(* CoDeSys 2.3.9.35 project: Сушка v1.1.pro *)
(* Libraries: IECSFC.LIB 13.4.06 15:51:28, ANALYZATION.LIB 5.10.99 09:05:06, Util.lib 18.5.10 15:14:28, STANDARD.LIB 4.10.05 11:14:46, SYSLIBTIME.LIB 20.2.06 13:31:16 *)

(* PLC configuration (modules and I/O channels)
Fast discrete inputs [I_SIMPLE_INPUT] node 0, in %IB0 out %QB0 {Filtrationtime = 10; Visibility = No}
  AT %IX0.0 [BitInput] Discrete input 1
  AT %IX0.1 [BitInput] Discrete input 2
Discrete inputs - 16 [ID130] node 1, in %IB1 out %QB1 {Filtrationtime_GeneralINP = 1; Visibility = No; PinCount = 16}
  AT %IB1.0 [ByteInput] 8 discrete inputs
  AT %IB1.1 [ByteInput] 8 discrete inputs
Fast discrete outputs [OWEN_ID570] node 2, in %IB2 out %QB2 {SafeValueBool = FALSE; SafeValueBool = FALSE; SafeValueBool = FALSE; SafeValueBool = FALSE; Visibility = No}
  AT %QX2.0 [BitOutput] Fast discrete output 1
  AT %QX2.1 [BitOutput] Fast discrete output 2
  AT %QX2.2 [BitOutput] Fast discrete output 3
  AT %QX2.3 [BitOutput] Fast discrete output 4
Discrete outputs - 8 [ID131] node 3, in %IB3 out %QB3 {SafeValueByte = 0; Visibility = No; PinCount = 10}
  AT %QB3.0 [ByteOutput] 8 discrete outputs
Special input [ID103] node 4, in %IB4 out %QB4 {Filtrationtime = 1000; PinCount = 1; WatchDogPeriod = 400; PollPeriod = 3000; Visibility = No}
  AT %IX4.0 [BitInput] Special input
Special output [ID104] node 5, in %IB5 out %QB5 {Visibility = No; PinCount = 1}
  AT %QX5.0 [BitOutput] Special output
AT %QD6.0 [DWordOutput] Last address
AT %QW6.1 [WordOutput] Last error
RS-485-1 [COM1_USART] node 0, in %IB6.0 out %QB6.0 {CommunicationSpeed = 9600; Parity = NO PARITY CHECK; BitLength = 8 bits; StopLength = One stop bit; InterfaceType = RS485; FrameOriented = RTU; Timeout = 0; Visibility = No}
AT %QB6.1.0 [ComChannel] Command (0xff - Start)
AT %IW6.1.0.0 [WordInput]
AT %IW6.1.1.0 [WordInput]
AT %IW6.1.2.0 [WordInput]
Button [ID003] node 7, in %IB7 out %QB7
  AT %IX7.0 [BitInput] Button Start/Stop
RS-485-2 [COM3_USART] node 0, in %IB8.0.0 out %QB8.0.0 {CommunicationSpeed = 11520; Parity = NO PARITY CHECK; BitLength = 8 bits; StopLength = One stop bit; InterfaceType = RS232; FrameOriented = RTU; Timeout = 0; Visibility = No}
TCP [TCP_ID221] node 1, in %IB8.0.1 out %QB8.0.1 {RemotePort = 502; Visibility = No}
2 byte [Register] node 1, in %IB8.1 out %QB8.1
  AT %QW8.1.0 [WordOutput]
2 byte [Register] node 2, in %IB8.2 out %QB8.2
  AT %QW8.2.0 [WordOutput]
2 byte [Register] node 3, in %IB8.3 out %QB8.3
  AT %QW8.3.0 [WordOutput]
2 byte [Register] node 4, in %IB8.4 out %QB8.4
  AT %QW8.4.0 [WordOutput]
2 byte [Register] node 5, in %IB8.5 out %QB8.5
  AT %QW8.5.0 [WordOutput]
2 byte [Register] node 6, in %IB8.6 out %QB8.6
  AT %QW8.6.0 [WordOutput]
2 byte [Register] node 7, in %IB8.7 out %QB8.7
  AT %QW8.7.0 [WordOutput]
2 byte [Register] node 8, in %IB8.8 out %QB8.8
  AT %QW8.8.0 [WordOutput]
2 byte [Register] node 9, in %IB8.9 out %QB8.9
  AT %QW8.9.0 [WordOutput]
2 byte [Register] node 10, in %IB8.10 out %QB8.10
  AT %QW8.10.0 [WordOutput]
2 byte [Register] node 11, in %IB8.11 out %QB8.11
  AT %QW8.11.0 [WordOutput]
2 byte [Register] node 12, in %IB8.12 out %QB8.12
  AT %QW8.12.0 [WordOutput]
2 byte [Register] node 13, in %IB8.13 out %QB8.13
  AT %QW8.13.0 [WordOutput]
2 byte [Register] node 14, in %IB8.14 out %QB8.14
  AT %QW8.14.0 [WordOutput]
2 byte [Register] node 15, in %IB8.15 out %QB8.15
  AT %QW8.15.0 [WordOutput]
2 byte [Register] node 16, in %IB8.16 out %QB8.16
  AT %QW8.16.0 [WordOutput]
2 byte [Register] node 17, in %IB8.17 out %QB8.17
  AT %QW8.17.0 [WordOutput]
2 byte [Register] node 18, in %IB8.18 out %QB8.18
  AT %QW8.18.0 [WordOutput]
2 byte [Register] node 19, in %IB8.19 out %QB8.19
  AT %QW8.19.0 [WordOutput]
2 byte [Register] node 20, in %IB8.20 out %QB8.20
  AT %QW8.20.0 [WordOutput]
  AT %QW8.21.0 [WordOutput]
  AT %QW8.22.0 [WordOutput]
  AT %QW8.23.0 [WordOutput]
  AT %QW8.24.0 [WordOutput]
  AT %QW8.25.0 [WordOutput]
  AT %QW8.26.0 [WordOutput]
AT %QB8.27.0 [ByteOutput]
AT %QW8.28.0 [WordOutput]
AT %QW8.29.0 [WordOutput]
AT %QW8.30.0 [WordOutput]
AT %QW8.31.0 [WordOutput]
*)

(* POU PLC_PRG, LD *)
PROGRAM PLC_PRG
VAR
(* Блок часов реального времени*)
	get_time: t_n_d;
	outSecond: WORD;
	outMinute AT %QW8.26.0: WORD;
	outHour AT %QW8.25.0: WORD;
	outDay AT %QW8.24.0: WORD;
	outMonth AT %QW8.13.0: WORD;
	outYear AT %QW8.14.0: WORD;
	outDayOfWeek: WORD;
(*Насторойка часов реального времени*)
	inMin AT %QW8.10.0:WORD;
	inHour AT %QW8.11.0:WORD;
	inday AT %QW8.12.0:WORD;
(*Команда на старт определенной печи по заданному времени*)
	Start1: BOOL;
	Start2: BOOL;
	Start3: BOOL;
(*Команда на остановку определенной печи через промежуток времени, заданный оператором*)
	stop1: BOOL;
	stop2: BOOL;
	stop3: BOOL;
(*Блоки-регуляторы включения\отключения вентиляторов и тенов, в зависимости от темпреатуры*)
	HYST1: HYSTERESIS;
	min_temp1: WORD;
	max_temp1: WORD;
	out1: BOOL;
	HYST2: HYSTERESIS;
	max_temp2: WORD;
	min_temp2: WORD;
	out2: BOOL;
	HYST3: HYSTERESIS;
	max_temp3: WORD;
	min_temp3: WORD;
	out3: BOOL;
(*Блоки задания на влючение, в зависимости от реального времени*)
	set_time_start1: s_t_s;
	set_time_start2: s_t_s;
	set_time_start3: s_t_s;
(*Продолжительность сушки после достижения номинальной температуры*)
	time_stop1: t_stop;
	time_stop2: t_stop;
	time_stop3: t_stop;
(*Входящая температура*)
	in_temp1 AT %IW6.1.0.0: WORD;
	in_temp2 AT %IW6.1.1.0: WORD;
	in_temp3 AT %IW6.1.2.0: WORD;
(*Блок для упрощения схемы*)
	min_max: min_max;
(*Выходные сигналы для управления вентиляторами и тенами*)
	vent1 AT %QX2.3: BOOL;
	vent2 AT %QX3.0.1: BOOL;
	vent3 AT %QX3.0.3: BOOL;

	ten1 AT %QX2.2: BOOL;
	ten2 AT %QX3.0.0: BOOL;
	ten3 AT %QX3.0.2: BOOL;

	ton1: TON;
	ton2: TON;
	ton3: TON;

(*Входной переключатель автомат/ручное*)
	in_switch1 AT %IX0.0:BOOL;
(*Выходное отображение автомат/ручное*)
	in_sw1 AT %QX8.27.0.0:BOOL;
(*Выходящая температура для отображения*)
	out_temp1 AT %QW8.21.0: WORD;
	out_temp2 AT %QW8.22.0: WORD;
	out_temp3 AT %QW8.23.0: WORD;
(*Параметры вносимые оператором для блока задания на влючение печи сушки №1*)
	Hour_IP1 AT %QW8.1.0: WORD;
	Minute_IP1 AT %QW8.2.0: WORD;
	Day_IP1 AT %QW8.3.0: WORD;
(*Параметры вносимые оператором для блока задания на влючение печи сушки №2*)
	Hour_IP2 AT %QW8.4.0: WORD;
	Minute_IP2 AT %QW8.5.0: WORD;
	Day_IP2 AT %QW8.6.0: WORD;
(*Параметры вносимые оператором для блока задания на влючение печи сушки №3*)
	Hour_IP3 AT %QW8.7.0: WORD;
	Minute_IP3 AT %QW8.8.0: WORD;
	Day_IP3 AT %QW8.9.0: WORD;
(*Время работы, вносимые оператором для печей сушек №1,2,3*)
	work_time1 AT %QW8.15.0: WORD;
	work_time2 AT %QW8.16.0: WORD;
	work_time3 AT %QW8.17.0: WORD;
(*Уставки температуры, вносимые оператором для печей сушек №1,2,3*)
	set_temp1 AT %QW8.18.0: WORD;
	set_temp2 AT %QW8.19.0: WORD;
	set_temp3 AT %QW8.20.0: WORD;
(*Выходное отображение старта системы*)
	Start11 AT %QX8.27.0.1: BOOL;
	Start22 AT %QX8.27.0.2: BOOL;
	Start33 AT %QX8.27.0.3: BOOL;
(*Кнопка подтверддения пуска*)
	but_in1 AT %QW8.28.0:WORD;
	but1: BOOL;
	but_in2 AT %QW8.29.0:WORD;
	but2: BOOL;
	but_in3 AT %QW8.30.0:WORD;
	but3: BOOL;
(*Кнопка "Грибок"*)
	stop_grib AT %IX0.1: BOOL;
(*Контроль аварийного привышения температуры в камерах сушил №1,2,3*)
	av_1 AT %IX1.0.0: BOOL;
	av_2 AT %IX1.0.1: BOOL;
	av_3 AT %IX1.0.2: BOOL;
(*Коменда установки значений RTC*)
	set_t:BOOL;
(*Выходное реле выбора режима работы*)
	avto_ruch AT %QX2.1: BOOL;
(*Блок остановки программы по приходу нуля из Scada&*)
	stop_if: stop_if;
	st_if1: BOOL;
	st_if2: BOOL;
	st_if3: BOOL;

	set_time AT %QW8.31.0: WORD;
END_VAR
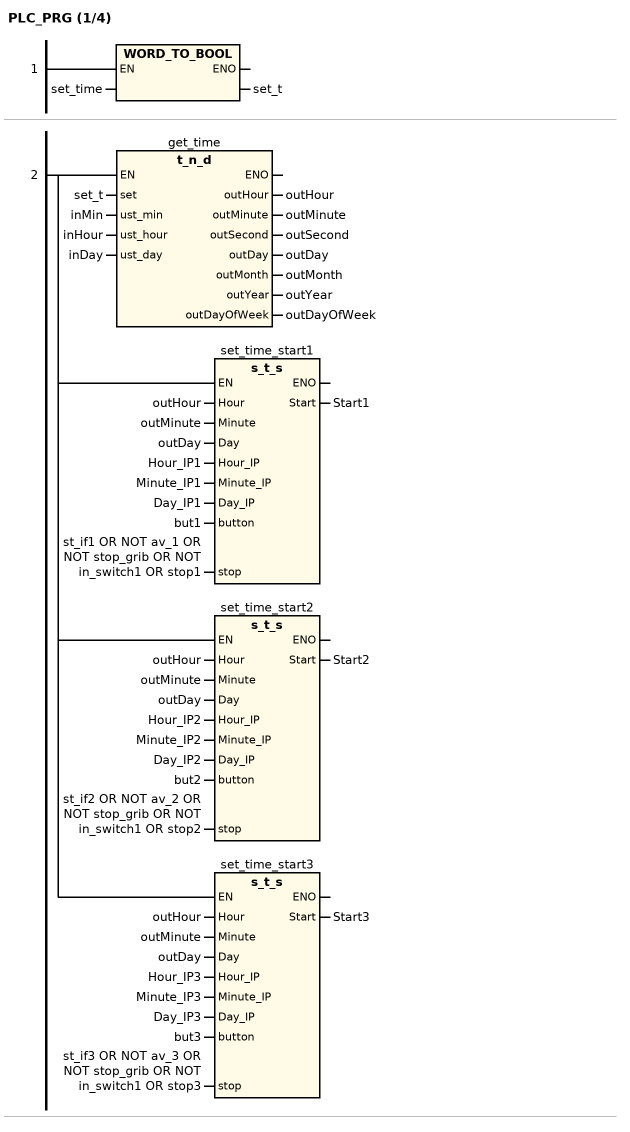
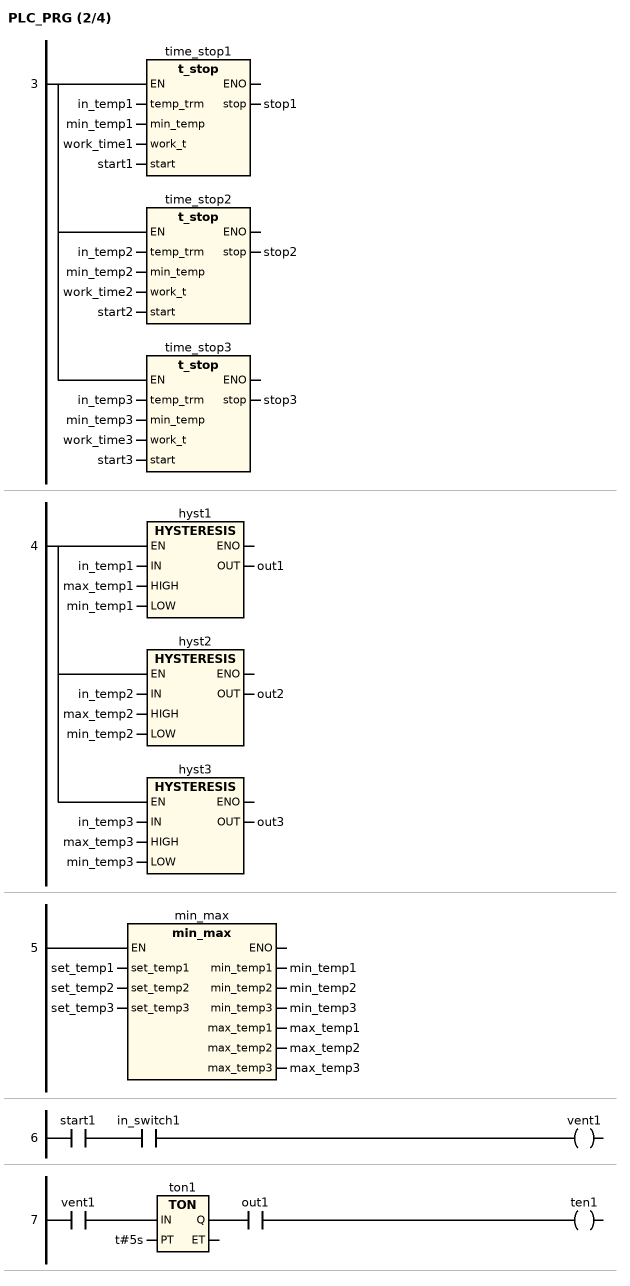
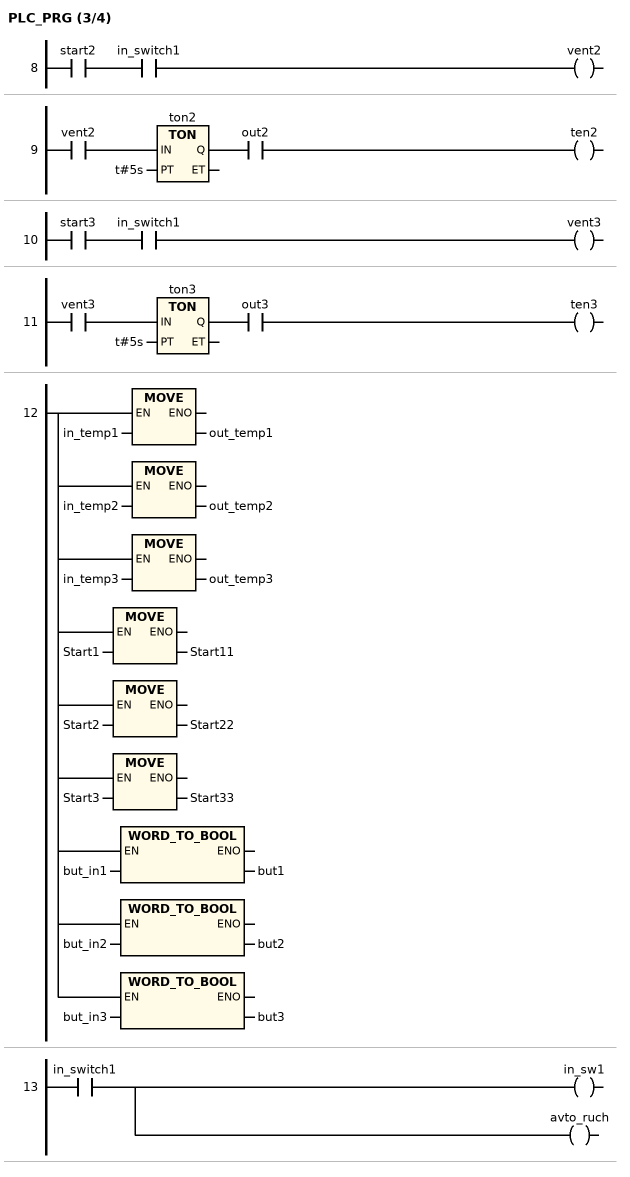
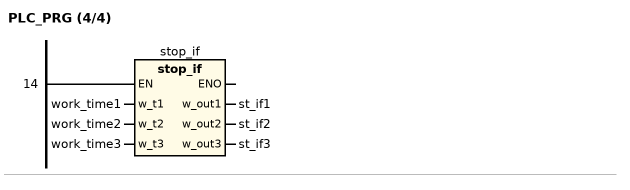
_LD_ (* Ladder Diagram *)
NETWORK 1
	*
		EN --- WORD_TO_BOOL(set_time) => set_t
NETWORK 2
	*
		EN --- get_time:t_n_d(set: set_t, ust_min: inMin, ust_hour: inHour, ust_day: inDay, outMinute => outMinute, outSecond => outSecond, outDay => outDay, outMonth => outMonth, outYear => outYear, outDayOfWeek => outDayOfWeek) => outHour
		EN --- set_time_start1:s_t_s(Hour: outHour, Minute: outMinute, Day: outDay, Hour_IP: Hour_IP1, Minute_IP: Minute_IP1, Day_IP: Day_IP1, button: but1, stop: st_if1 OR NOT av_1 OR NOT stop_grib OR NOT in_switch1 OR stop1) => Start1
		EN --- set_time_start2:s_t_s(Hour: outHour, Minute: outMinute, Day: outDay, Hour_IP: Hour_IP2, Minute_IP: Minute_IP2, Day_IP: Day_IP2, button: but2, stop: st_if2 OR NOT av_2 OR NOT stop_grib OR NOT in_switch1 OR stop2) => Start2
		EN --- set_time_start3:s_t_s(Hour: outHour, Minute: outMinute, Day: outDay, Hour_IP: Hour_IP3, Minute_IP: Minute_IP3, Day_IP: Day_IP3, button: but3, stop: st_if3 OR NOT av_3 OR NOT stop_grib OR NOT in_switch1 OR stop3) => Start3
NETWORK 3
	*
		EN --- time_stop1:t_stop(temp_trm: in_temp1, min_temp: min_temp1, work_t: work_time1, start: start1) => stop1
		EN --- time_stop2:t_stop(temp_trm: in_temp2, min_temp: min_temp2, work_t: work_time2, start: start2) => stop2
		EN --- time_stop3:t_stop(temp_trm: in_temp3, min_temp: min_temp3, work_t: work_time3, start: start3) => stop3
NETWORK 4
	*
		EN --- hyst1:HYSTERESIS(IN: in_temp1, HIGH: max_temp1, LOW: min_temp1) => out1
		EN --- hyst2:HYSTERESIS(IN: in_temp2, HIGH: max_temp2, LOW: min_temp2) => out2
		EN --- hyst3:HYSTERESIS(IN: in_temp3, HIGH: max_temp3, LOW: min_temp3) => out3
NETWORK 5
	*
		EN --- min_max:min_max(set_temp1: set_temp1, set_temp2: set_temp2, set_temp3: set_temp3, min_temp2 => min_temp2, min_temp3 => min_temp3, max_temp1 => max_temp1, max_temp2 => max_temp2, max_temp3 => max_temp3) => min_temp1
NETWORK 6
	[start1] - [in_switch1] --- (vent1)
NETWORK 7
	[vent1] - ton1:TON(IN: *, PT: t#5s) - [out1] --- (ten1)
NETWORK 8
	[start2] - [in_switch1] --- (vent2)
NETWORK 9
	[vent2] - ton2:TON(IN: *, PT: t#5s) - [out2] --- (ten2)
NETWORK 10
	[start3] - [in_switch1] --- (vent3)
NETWORK 11
	[vent3] - ton3:TON(IN: *, PT: t#5s) - [out3] --- (ten3)
NETWORK 12
	*
		EN --- MOVE(in_temp1) => out_temp1
		EN --- MOVE(in_temp2) => out_temp2
		EN --- MOVE(in_temp3) => out_temp3
		EN --- MOVE(Start1) => Start11
		EN --- MOVE(Start2) => Start22
		EN --- MOVE(Start3) => Start33
		EN --- WORD_TO_BOOL(but_in1) => but1
		EN --- WORD_TO_BOOL(but_in2) => but2
		EN --- WORD_TO_BOOL(but_in3) => but3
NETWORK 13
	[in_switch1] --- (in_sw1) (avto_ruch)
NETWORK 14
	*
		EN --- stop_if:stop_if(w_t1: work_time1, w_t2: work_time2, w_t3: work_time3, w_out2 => st_if2, w_out3 => st_if3) => st_if1
_END_LD_
(* the same logic as Structured Text *)
(* Network 1 *)
set_t := WORD_TO_BOOL(set_time);
(* Network 2 *)
get_time(set := set_t, ust_min := inMin, ust_hour := inHour, ust_day := inDay);
outMinute := get_time.outMinute;
outSecond := get_time.outSecond;
outDay := get_time.outDay;
outMonth := get_time.outMonth;
outYear := get_time.outYear;
outDayOfWeek := get_time.outDayOfWeek;
outHour := get_time.outHour;
set_time_start1(Hour := outHour, Minute := outMinute, Day := outDay, Hour_IP := Hour_IP1, Minute_IP := Minute_IP1, Day_IP := Day_IP1, button := but1, stop := st_if1 OR NOT av_1 OR NOT stop_grib OR NOT in_switch1 OR stop1);
Start1 := set_time_start1.Start;
set_time_start2(Hour := outHour, Minute := outMinute, Day := outDay, Hour_IP := Hour_IP2, Minute_IP := Minute_IP2, Day_IP := Day_IP2, button := but2, stop := st_if2 OR NOT av_2 OR NOT stop_grib OR NOT in_switch1 OR stop2);
Start2 := set_time_start2.Start;
set_time_start3(Hour := outHour, Minute := outMinute, Day := outDay, Hour_IP := Hour_IP3, Minute_IP := Minute_IP3, Day_IP := Day_IP3, button := but3, stop := st_if3 OR NOT av_3 OR NOT stop_grib OR NOT in_switch1 OR stop3);
Start3 := set_time_start3.Start;
(* Network 3 *)
time_stop1(temp_trm := in_temp1, min_temp := min_temp1, work_t := work_time1, start := start1);
stop1 := time_stop1.stop;
time_stop2(temp_trm := in_temp2, min_temp := min_temp2, work_t := work_time2, start := start2);
stop2 := time_stop2.stop;
time_stop3(temp_trm := in_temp3, min_temp := min_temp3, work_t := work_time3, start := start3);
stop3 := time_stop3.stop;
(* Network 4 *)
hyst1(IN := in_temp1, HIGH := max_temp1, LOW := min_temp1);
out1 := hyst1.OUT;
hyst2(IN := in_temp2, HIGH := max_temp2, LOW := min_temp2);
out2 := hyst2.OUT;
hyst3(IN := in_temp3, HIGH := max_temp3, LOW := min_temp3);
out3 := hyst3.OUT;
(* Network 5 *)
min_max(set_temp1 := set_temp1, set_temp2 := set_temp2, set_temp3 := set_temp3);
min_temp2 := min_max.min_temp2;
min_temp3 := min_max.min_temp3;
max_temp1 := min_max.max_temp1;
max_temp2 := min_max.max_temp2;
max_temp3 := min_max.max_temp3;
min_temp1 := min_max.min_temp1;
(* Network 6 *)
vent1 := start1 AND in_switch1;
(* Network 7 *)
ton1(IN := vent1, PT := t#5s);
ten1 := ton1.Q AND out1;
(* Network 8 *)
vent2 := start2 AND in_switch1;
(* Network 9 *)
ton2(IN := vent2, PT := t#5s);
ten2 := ton2.Q AND out2;
(* Network 10 *)
vent3 := start3 AND in_switch1;
(* Network 11 *)
ton3(IN := vent3, PT := t#5s);
ten3 := ton3.Q AND out3;
(* Network 12 *)
out_temp1 := in_temp1;
out_temp2 := in_temp2;
out_temp3 := in_temp3;
Start11 := Start1;
Start22 := Start2;
Start33 := Start3;
but1 := WORD_TO_BOOL(but_in1);
but2 := WORD_TO_BOOL(but_in2);
but3 := WORD_TO_BOOL(but_in3);
(* Network 13 *)
in_sw1 := in_switch1;
avto_ruch := in_switch1;
(* Network 14 *)
stop_if(w_t1 := work_time1, w_t2 := work_time2, w_t3 := work_time3);
st_if2 := stop_if.w_out2;
st_if3 := stop_if.w_out3;
st_if1 := stop_if.w_out1;
END_PROGRAM

(* POU t_n_d, ST *)
FUNCTION_BLOCK t_n_d
VAR
	GetTime: CurTimeEx;
	TimeAndDate: SystemTimeDate;
	Sys_Time: SysTime64;
END_VAR

VAR_INPUT
	set: BOOL;
	ust_min:WORD;
	ust_hour:WORD;
	ust_day:WORD;
END_VAR

VAR_OUTPUT
	outHour: WORD;
	outMinute: WORD;
	outSecond: WORD;
	outDay: WORD;
	outMonth: WORD;
	outYear: WORD;
	outDayOfWeek: WORD;
END_VAR
(*Текущее время*)
	TimeAndDate.Day :=0;
	TimeAndDate.DayOfWeek :=0;
	TimeAndDate.dwHighMsec :=0;
	TimeAndDate.dwLowMSecs :=0;
	TimeAndDate.Milliseconds :=0;
	TimeAndDate.Minute :=0;
	TimeAndDate.Second :=0;
	TimeAndDate.Hour :=0;
	TimeAndDate.Year :=0;
	TimeAndDate.Month :=0;
	Sys_time.ulHigh :=0;
	Sys_time.ulLow :=0;
	GetTime (SystemTime:=Sys_Time , TimeDate:= TimeAndDate);

IF set THEN
	TimeAndDate.Day :=ust_day;
	TimeAndDate.Minute :=ust_min;
	TimeAndDate.Hour :=ust_hour;
	GetTime (SystemTime:=Sys_Time , TimeDate:= TimeAndDate);
END_IF

	outSecond:=TimeAndDate.Second;
	outMinute:=TimeAndDate.Minute;
	outHour:=TimeAndDate.Hour;
	outDay:=TimeAndDate.Day;
	outMonth:=TimeAndDate.Month;
	outYear:=TimeAndDate.Year;
	outDayOfWeek:=TimeAndDate.DayOfWeek;

(*	outdwHighMsec:=TimeAndDate.dwHighMsec;
	outdwLowMSecs:=TimeAndDate.dwLowMSecs;*)

(*	outulHigh:=Sys_time.ulHigh;
	outulLow:=Sys_time.ulLow;*)
END_FUNCTION_BLOCK

(* POU s_t_s, LD *)
FUNCTION_BLOCK s_t_s

VAR_INPUT
	Hour: WORD;
	Minute: WORD;
	Day: WORD;
	Hour_IP: WORD;
	Minute_IP: WORD;
	Day_IP: WORD;
	button: BOOL;
	stop: BOOL;
END_VAR
VAR
	set_hour: BOOL;
	set_min: BOOL;
	set_day: BOOL;
	r_t: R_TRIG;
	pr1: BOOL;
	pr2: BOOL;
END_VAR
VAR_OUTPUT
	Start: BOOL;
END_VAR
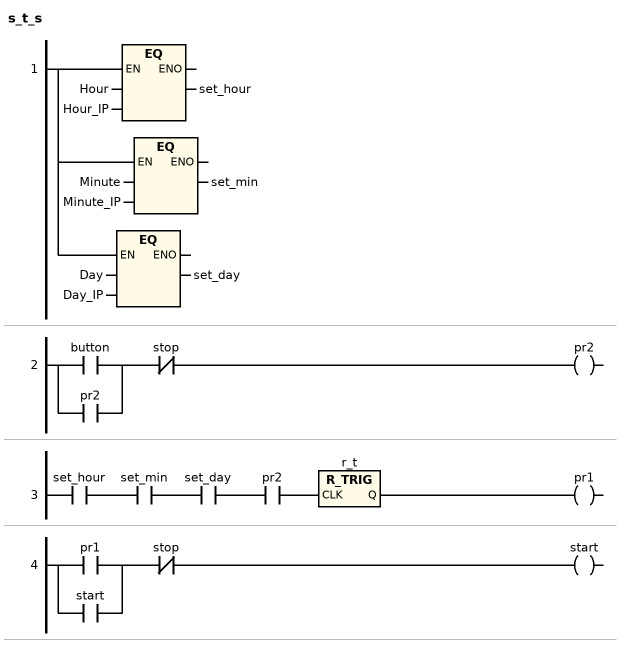
_LD_ (* Ladder Diagram *)
NETWORK 1
	*
		EN --- EQ(Hour, Hour_IP) => set_hour
		EN --- EQ(Minute, Minute_IP) => set_min
		EN --- EQ(Day, Day_IP) => set_day
NETWORK 2
	{ [button] | [pr2] } - [/stop] --- (pr2)
NETWORK 3
	[set_hour] - [set_min] - [set_day] - [pr2] - r_t:R_TRIG(CLK: *) --- (pr1)
NETWORK 4
	{ [pr1] | [start] } - [/stop] --- (start)
_END_LD_
(* the same logic as Structured Text *)
(* Network 1 *)
set_hour := Hour = Hour_IP;
set_min := Minute = Minute_IP;
set_day := Day = Day_IP;
(* Network 2 *)
pr2 := (button OR pr2) AND NOT stop;
(* Network 3 *)
r_t(CLK := set_hour AND set_min AND set_day AND pr2);
pr1 := r_t.Q;
(* Network 4 *)
start := (pr1 OR start) AND NOT stop;
END_FUNCTION_BLOCK

(* POU t_stop, LD *)
FUNCTION_BLOCK t_stop
VAR_INPUT
	temp_trm: WORD;
	min_temp: WORD;
	work_t: WORD;
	start: BOOL;
END_VAR
VAR
	c_s: BOOL;
	T1: DWORD;
	w_t: TIME;
	stop_work: TON;
	str: BOOL;
	pr1: BOOL;
END_VAR

VAR_OUTPUT
	stop: BOOL;
END_VAR
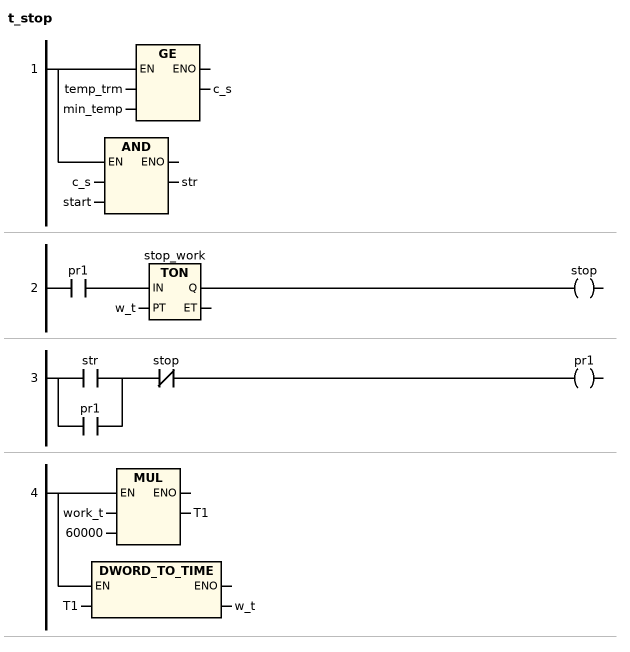
_LD_ (* Ladder Diagram *)
NETWORK 1
	*
		EN --- GE(temp_trm, min_temp) => c_s
		EN --- AND(c_s, start) => str
NETWORK 2
	[pr1] - stop_work:TON(IN: *, PT: w_t) --- (stop)
NETWORK 3
	{ [str] | [pr1] } - [/stop] --- (pr1)
NETWORK 4
	*
		EN --- MUL(work_t, 60000) => T1
		EN --- DWORD_TO_TIME(T1) => w_t
_END_LD_
(* the same logic as Structured Text *)
(* Network 1 *)
c_s := temp_trm >= min_temp;
str := c_s AND start;
(* Network 2 *)
stop_work(IN := pr1, PT := w_t);
stop := stop_work.Q;
(* Network 3 *)
pr1 := (str OR pr1) AND NOT stop;
(* Network 4 *)
T1 := work_t * 60000;
w_t := DWORD_TO_TIME(T1);
END_FUNCTION_BLOCK

(* POU min_max, LD *)
FUNCTION_BLOCK min_max

VAR_INPUT
	set_temp1:WORD;
	set_temp2:WORD;
	set_temp3:WORD;
END_VAR

VAR_OUTPUT
	min_temp1:WORD;
	min_temp2:WORD;
	min_temp3:WORD;
	max_temp1:WORD;
	max_temp2:WORD;
	max_temp3:WORD;
END_VAR
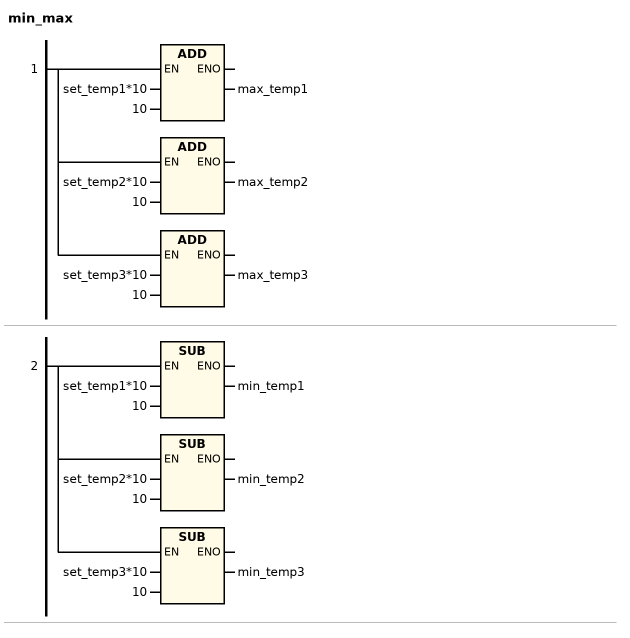
_LD_ (* Ladder Diagram *)
NETWORK 1
	*
		EN --- ADD(set_temp1*10, 10) => max_temp1
		EN --- ADD(set_temp2*10, 10) => max_temp2
		EN --- ADD(set_temp3*10, 10) => max_temp3
NETWORK 2
	*
		EN --- SUB(set_temp1*10, 10) => min_temp1
		EN --- SUB(set_temp2*10, 10) => min_temp2
		EN --- SUB(set_temp3*10, 10) => min_temp3
_END_LD_
(* the same logic as Structured Text *)
(* Network 1 *)
max_temp1 := (set_temp1*10) + 10;
max_temp2 := (set_temp2*10) + 10;
max_temp3 := (set_temp3*10) + 10;
(* Network 2 *)
min_temp1 := (set_temp1*10) - 10;
min_temp2 := (set_temp2*10) - 10;
min_temp3 := (set_temp3*10) - 10;
END_FUNCTION_BLOCK

(* POU stop_if, ST *)
FUNCTION_BLOCK stop_if
VAR_INPUT
	w_t1:WORD;
	w_t2:WORD;
	w_t3:WORD;
END_VAR

VAR_OUTPUT
	w_out1:BOOL;
	w_out2:BOOL;
	w_out3:BOOL;
END_VAR
IF w_t1=0
THEN w_out1:=TRUE;
ELSE w_out1:=FALSE;
END_IF

IF w_t2=0
THEN w_out2:=TRUE;
ELSE w_out2:=FALSE;
END_IF

IF w_t3=0
THEN w_out3:=TRUE;
ELSE w_out3:=FALSE;
END_IF
END_FUNCTION_BLOCK
